FUNCTION IEEE32_TO_REAL : REAL
VAR_INPUT
	IN:DWORD;
END_VAR
VAR
	PTREAL:POINTER TO REAL;
END_VAR

PTREAL:=ADR(IN);
IEEE32_TO_REAL:=PTREAL^;

END_FUNCTION

(* stored: Version 1.1.0.1, ProductVersion 3.1.4024.9
   POU IEEE32_TO_REAL: Id {0ad90c61-97e8-4bd6-bbc7-678ff1cf5421}, SpecialFunc None *)
